// TIA Portal V17 export
// export: Created 2024-09-02T12:50:36.4832913Z, ExportSetting WithDefaults, DisplayName Totally Integrated Automation Portal, DisplayVersion V17, DisplayName TIA Portal Openness, DisplayVersion V17, DisplayName TIA Portal Version Control Interface, DisplayVersion V17, DisplayName STEP 7 Professional, DisplayVersion V17, DisplayName STEP 7 Safety, DisplayVersion V17, DisplayName WinCC Professional, DisplayVersion V17
TYPE "TypeMobyQDS_1"
// stored: IsFailsafeCompliant false
   STRUCT
      WERT : Array[1..30] of Byte;
   END_STRUCT;
END_TYPE
